Staubli VAL3: GasChoose.pgx

public program GasChoose(num x_nGasIndex)
begin
  //2015.05.28
  //气体选择，为特定的气体做选择


  if roundDown(x_nGasIndex)!=roundUp(x_nGasIndex)
      x_nGasIndex=0
  endIf


  switch  x_nGasIndex
    case 0
      dDio["UsO_bNull5"]=false
      dDio["UsO_bNull6"]=false
      dDio["UsO_bNull8"]=false

    break

    case 1
      dDio["UsO_bNull5"]=true
      dDio["UsO_bNull6"]=false
      dDio["UsO_bNull8"]=false
    break


    case 2
      dDio["UsO_bNull5"]=false
      dDio["UsO_bNull6"]=true
      dDio["UsO_bNull8"]=false
    break


    case 3
      dDio["UsO_bNull5"]=false
      dDio["UsO_bNull6"]=false
      dDio["UsO_bNull8"]=true

    break





  endSwitch

  call Digtal2Analog()






end
